FUNCTION_BLOCK LinearContinuousDrive_3Sensor EXTENDS FBA_LinearDrive IMPLEMENTS I_LinearContinuousDrive
VAR_INPUT
	drive : I_ContinuousDrive;
	allowDualSideTraverse : BOOL; //allows motion between home to retractLimit
END_VAR
VAR
	extendLimit AT %I* : BOOL;
	retractLimit AT %I* : BOOL;
END_VAR

override();

ready := bEnable AND NOT Active AND HomeSet;

PROPERTY Active : BOOL
GET
Active := drive.Active;
END_GET
END_PROPERTY

PROPERTY AtExtendLimit : BOOL
GET
AtExtendLimit := extendLimit <> sensorDefaultState;
END_GET
END_PROPERTY

PROPERTY AtRetractLimit : BOOL
GET
AtRetractLimit := retractLimit <> sensorDefaultState;
END_GET
END_PROPERTY

PROPERTY Error : BOOL
GET
error := drive.Error;
END_GET
END_PROPERTY

METHOD homingSequence : BOOL
(*
homing sequence is different for linear motion devices with limit sensors
*)
CASE step OF
	Homing.IDLE:
		reset();
		IF bEnable THEN
			step := Homing.RETRY;
		END_IF
		
	Homing.START:
		IF AtHome THEN
			step := Homing.STOP;
			
		ELSIF AtRetractLimit THEN
			step := Homing.RETRY;
			
		ELSE
			moveContinuous(newDirection:= MC_Positive_Direction);
		END_IF
		
	Homing.RETRY:
		IF AtExtendLimit THEN
			step := Homing.START;
		ELSE
			moveContinuous(newDirection:= MC_Positive_Direction);
		END_IF
		
	Homing.STOP:
		IF stop() THEN
			step := Homing.DONE;
		END_IF
		
	Homing.DONE:
		homingComplete := TRUE;
		step := Homing.IDLE;
		
END_CASE
END_METHOD

METHOD moveContinuous : BOOL
VAR_INPUT
	newDirection : MC_Direction;
END_VAR
drive.moveContinuous(newDirection:= newDirection);

direction := newDirection;
END_METHOD

METHOD PRIVATE override : BOOL
VAR_INPUT
END_VAR
(*
-at home and attempting to traverse outward
-at outer limit and attempting to traverse outward
-at inner limit and attempting to traverse inwards
*)
(*
inward = negative direction, negative velocity
outward = positive direction, positive velocity
*)

IF error THEN
	stop();
	reset();
	
ELSIF
	(NOT allowDualSideTraverse AND AtHome AND direction = MC_Positive_Direction) OR
	(AtExtendLimit AND direction = MC_Negative_Direction) OR
	(AtRetractLimit AND direction = MC_Positive_Direction)
THEN
	stop();
END_IF
END_METHOD

METHOD reset : BOOL
VAR_INPUT
END_VAR
reset := drive.reset();
END_METHOD

METHOD stop : BOOL
VAR_INPUT
END_VAR
stop := drive.stop();
END_METHOD

METHOD toHome : BOOL
VAR_INPUT
END_VAR
IF AtHome THEN
	toHome := TRUE;
ELSE
	moveContinuous(newDirection := MC_Negative_Direction);
END_IF
END_METHOD

END_FUNCTION_BLOCK

(* stored: Version 1.1.0.1, ProductVersion 3.1.4024.11
   POU LinearContinuousDrive_3Sensor: Id {c467e44f-af63-4286-b82b-3e7ba5ea1767}, SpecialFunc None
   Folder Private: Id {d211720d-bf33-43c2-b97b-9bc460002af6}
   Folder Properties: Id {4c069781-4249-4308-bc50-af0d70330c8a}
   Property Active: Id {bf5d36bc-a4f2-42dd-b0ac-8f5c59df6a46}
   Get Get: Id {6e80628a-fc35-44c5-9092-9b335c9cf43d}
   Property AtExtendLimit: Id {8c293064-3fc1-4d9f-89fa-66291c82c6e4}
   Get Get: Id {38ef1b4a-30e7-40ef-9d6f-7a4281365446}
   Property AtRetractLimit: Id {6e7c4787-d411-44a8-b293-7c2c2db6c88a}
   Get Get: Id {9b1bda46-be46-4863-9580-8efee15dd0ab}
   Property Error: Id {ee5938c4-e4f1-4337-b19f-af6b44b7e68c}
   Get Get: Id {afe1da99-63d7-4c37-9430-508a695c342e}
   Method homingSequence: Id {ffedb226-e0f3-4c38-8967-7a54d726dcb1}
   Method moveContinuous: Id {754f0fff-2844-4cd6-8b0b-18a730ba41ee}
   Method override: Id {b3f9c944-3e9d-41d5-9c2b-556bbde52111}
   Method reset: Id {1dfe8ba1-7219-437d-bacb-f698ffd0f114}
   Method stop: Id {93e337fb-7d07-4a4f-96cf-77bfc5262acf}
   Method toHome: Id {1eecf68e-21ae-4160-8141-d818ea8d6c1f} *)
